// TIA Portal V17 export
// export: Created 2022-07-20T07:01:29.8821279Z, ExportSetting WithDefaults, DisplayName Totally Integrated Automation Portal, DisplayVersion V17, DisplayName TIA Portal Openness, DisplayVersion V17, DisplayName TIA Portal Version Control Interface, DisplayVersion V17, DisplayName SINAMICS Startdrive Advanced, DisplayVersion V17, DisplayName SINAMICS Startdrive G130, G150, S120, S150, SINAMICS MV, S210, DisplayVersion V17, DisplayName SINAMICS Startdrive G110M, G120, G120C, G120D, G120P, G115D, DisplayVersion V17, DisplayName STEP 7 Professional, DisplayVersion V17, DisplayName STEP 7 Safety, DisplayVersion V17, DisplayName WinCC Advanced, DisplayVersion V17
FUNCTION_BLOCK "FB10253_IfmLDH292"   // FB10253, LAD
{ S7_Optimized_Access := 'TRUE' }
VERSION : 0.1
// stored: AutoNumber false, IsIECCheckEnabled false, IsRetainMemResEnabled false, MemoryReserve 100, SetENOAutomatically false, UDAEnableTagReadback false
   VAR_OUTPUT
      CurrentHumidityPercentage : Real;
      CurrentTemperatureCelcius : Real;
   END_VAR
   VAR_IN_OUT
      ProcessDataWord_0 : Word;
      ProcessDataWord_2 : Word;
      ProcessDataWord_4 : Word;
      ProcessDataWord_5 : Word := 16#0;
   END_VAR
BEGIN

REGION Network 1 (SCL): Compute Humidity and Temperature
   IF (#ProcessDataWord_2.%B1 = 16#FF) THEN
       #CurrentHumidityPercentage := #ProcessDataWord_0 * 0.1;
   ELSE
       #CurrentHumidityPercentage := -1.0;
   END_IF;

   IF (#ProcessDataWord_5.%B1 = 16#FF) THEN
       #CurrentTemperatureCelcius := #ProcessDataWord_4 * 0.1;
   ELSE
       #CurrentHumidityPercentage := -1.0;
   END_IF;
END_REGION
END_FUNCTION_BLOCK
